FUNCTION_BLOCK CommFromMatlab1 (* Extracted Composite Function Block Type *)
  (* Version 5/20/2016, gulzha *)
  PACKAGE Main;
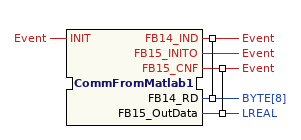
  EVENT_INPUT
    INIT; (* Initialization request event *)
  END_EVENT
  EVENT_OUTPUT
    FB14_IND WITH FB14_RD; (* Data read indication event *)
    FB15_INITO; (* Initialization Confirm *)
    FB15_CNF WITH FB15_OutData; (* Execution Confirmation *)
  END_EVENT
  VAR_OUTPUT
    FB14_RD : ARRAY [0..7] OF BYTE; (* Data read with every IND event *)
    FB15_OutData : LREAL;
  END_VAR
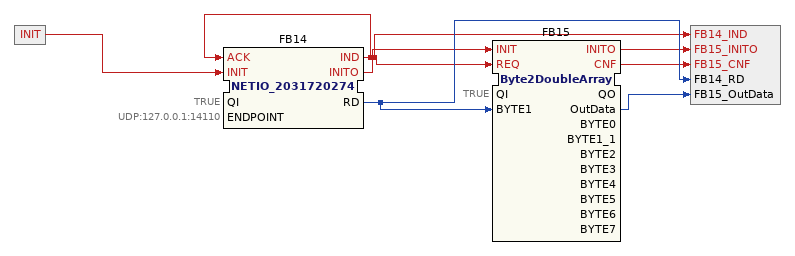
  FBS
    FB14 : NETIO_2031720274(QI := TRUE, ENDPOINT := UDP:127.0.0.1:14110); {SET_ATTRIBUTE(Configuration.GenericFBType.InterfaceParams, Runtime.IoCommon#I:=1;SD:BYTE[8];RD:BYTE[8])}
    FB15 : Byte2DoubleArray(QI := TRUE);
  END_FBS
  EVENT_CONNECTIONS
    FB14.IND TO FB14.ACK;
    FB14.IND TO FB15.REQ;
    FB14.INITO TO FB15.INIT;
    FB14.IND TO FB14_IND;
    FB15.INITO TO FB15_INITO;
    FB15.CNF TO FB15_CNF;
    INIT TO FB14.INIT;
  END_CONNECTIONS
  DATA_CONNECTIONS
    FB14.RD TO FB15.BYTE1;
    FB14.RD TO FB14_RD;
    FB15.OutData TO FB15_OutData;
  END_CONNECTIONS
END_FUNCTION_BLOCK
